// TIA Portal V19 export
VAR_GLOBAL   // PLC tag table "Default tag table"
   "HOOTER RESET" AT %Q0.0 : Bool;
   "EMERGENCY STOP" AT %I0.0 : Bool;
   "FRL LOW" AT %I0.1 : Bool;
   HOOTER AT %I0.2 : Bool;
   "MGF FEED PUMP P-101 A MCB TRIP" AT %I0.3 : Bool;
   "MGF FEED PUMP P-101 B MCB TRIP" AT %I0.4 : Bool;
   "MGF BACK WASH  P-102 A MCB TRIP" AT %I0.5 : Bool;
   "MGF BACK WASH P-102 B MCB TRIP" AT %I0.6 : Bool;
   "UF FEED PUMP P-103 A MCB TRIP" AT %I0.7 : Bool;
   "UF FEED PUMP P-103 B MCB TRIP" AT %I1.0 : Bool;
   "UF BLOWER AB-201 A MCB TRIP" AT %I1.1 : Bool;
   "UF BLOWER AB-201 B MCB TRIP" AT %I1.2 : Bool;
   "UF BACKWASH P-201A TRIP" AT %I1.3 : Bool;
   "UF BACKWASH P-201B TRIP" AT %I1.4 : Bool;
   SPARE_2 AT %I1.5 : Bool;
   "MGF FEED PUMP P-101 A" AT %Q0.1 : Bool;
   "MGF FEED PUMP P-101 B" AT %Q0.2 : Bool;
   "MGF BACK WASH P-102 A" AT %Q0.3 : Bool;
   "MGF BACK WASH P-102 B" AT %Q0.4 : Bool;
   "UF FEED PUMP P-103 A" AT %Q0.5 : Bool;
   "UF FEED PUMP P-103 B" AT %Q0.6 : Bool;
   "UF BLOWER AB-201 A" AT %Q0.7 : Bool;
   "UF BLOWER AB 201 B" AT %Q1.0 : Bool;
   "UF BACK WASH P-201 A" AT %Q1.1 : Bool;
   "SPARE(35)" AT %I8.0 : Bool;
   "SPARE(34)" AT %I8.1 : Bool;
   "DM FEED PUMP P-502 A MPCB TRIP" AT %I8.2 : Bool;
   "DM FEED PUMP P-502 B MPCB TRIP" AT %I8.3 : Bool;
   "DM FEED PUMP P-502 C MPCB TRIP" AT %I8.4 : Bool;
   "CIP P-601" AT %I8.5 : Bool;
   "BACK WASH RECOVERY P-801 A MPCB TRIP" AT %I8.6 : Bool;
   "BACK WASH RECOVERY P-801 B MPCB TRIP" AT %I8.7 : Bool;
   "ABFV-101 FEED BACK OPEN FEED BACK" AT %I9.0 : Bool;
   "ABFV-101 FEED BACK CLOSE FEED BACK" AT %I9.1 : Bool;
   "ABFV-102 FEED BACK OPEN FEED BACK" AT %I9.2 : Bool;
   "ABFV-102 FEED BACK CLOSE FEED BACK" AT %I9.3 : Bool;
   "ABFV-103 FEED BACK OPEN FEED BACK" AT %I9.4 : Bool;
   "ABFV-103 FEED BACK CLOSE FEED BACK" AT %I9.5 : Bool;
   "ABFV-104 FEED BACK OPEN FEED BACK" AT %I9.6 : Bool;
   "ABFV-104 FEED BACK CLOSE FEED BACK" AT %I9.7 : Bool;
   "UF BACK WASH  P-201 B" AT %Q8.0 : Bool;
   "DM FEED PUMP P-502 A" AT %Q8.1 : Bool;
   "DM FEED PUMP P-502 B" AT %Q8.2 : Bool;
   "DM FEED PUMP P-502 C" AT %Q8.3 : Bool;
   "CIP PUMP P-601" AT %Q8.4 : Bool;
   "BACK WASH RECOVERY P-801 A" AT %Q8.5 : Bool;
   "BACK WASH RECOVERY P-801 B" AT %Q8.6 : Bool;
   SPARE AT %Q8.7 : Bool;
   "SPARE(1)" AT %Q9.0 : Bool;
   "SPARE(2)" AT %Q9.1 : Bool;
   "DP-701" AT %Q9.2 : Bool;
   "DP-702" AT %Q9.3 : Bool;
   "NaOCL DOSING D-706 A" AT %Q9.4 : Bool;
   "NaOCL DOSING DP-706B" AT %Q9.5 : Bool;
   "ABFV-501" AT %Q9.6 : Bool;
   "ABFV-502" AT %Q9.7 : Bool;
   "ABFV 105 FEED BACK OPEN" AT %I12.0 : Bool;
   "ABFV 105 FEED BACK CLOSE" AT %I12.1 : Bool;
   "ABV 201 FEED BACK OPEN" AT %I12.2 : Bool;
   "ABV 201 FEED BACK CLOSE" AT %I12.3 : Bool;
   "ABFV 201 FEED BACK OPEN" AT %I12.4 : Bool;
   "ABFV 201 FEED BACK CLOSE" AT %I12.5 : Bool;
   "ABFV 202 FEED BACK OPEN" AT %I12.6 : Bool;
   "ABFV 202 FEED BACK CLOSE" AT %I12.7 : Bool;
   "ABFV 203 FEED BACK OPEN" AT %I13.0 : Bool;
   "ABFV 203 FEED BACK CLOSE" AT %I13.1 : Bool;
   "ABFV 204 FEED BACK OPEN" AT %I13.2 : Bool;
   "ABFV 204 FEED BACK CLOSE" AT %I13.3 : Bool;
   "ABFV 205 FEED BACK OPEN" AT %I13.4 : Bool;
   "ABFV 205 FEED BACK CLOSE" AT %I13.5 : Bool;
   "ABFV 206 FEED BACK OPEN" AT %I13.6 : Bool;
   "ABFV 206 FEED BACK CLOSE" AT %I13.7 : Bool;
   "ABFV 101 MULTIGRADE FILTER VALVE" AT %Q12.0 : Bool;
   "ABFV 102 MULTIGRADE FILTER VALVE" AT %Q12.1 : Bool;
   "ABFV 103 MULTIGRADE FILTER VALVE" AT %Q12.2 : Bool;
   "ABFV 104 MULTIGRADE FILTER VALVE" AT %Q12.3 : Bool;
   "ABFV 105 MULTIGRADE FILTER VALVE" AT %Q12.4 : Bool;
   "ABV 201 UF VALVE" AT %Q12.5 : Bool;
   "ABFV 201 UF VALVE" AT %Q12.6 : Bool;
   "ABFV 202 UF VALVE" AT %Q12.7 : Bool;
   "ABFV 203 UF VALVE" AT %Q13.0 : Bool;
   "ABFV 204 UF VALVE" AT %Q13.1 : Bool;
   "ABFV 205 UF VALVE" AT %Q13.2 : Bool;
   "ABFV 206 UF VALVE" AT %Q13.3 : Bool;
   "ABFV 207 UF VALVE" AT %Q13.4 : Bool;
   "ABFV 208 UF VALVE" AT %Q13.5 : Bool;
   "SPARE(3)" AT %Q13.6 : Bool;
   "SPARE(4)" AT %Q13.7 : Bool;
   "P-502 C ON" AT %I16.0 : Bool;
   "P-601 ON" AT %I16.1 : Bool;
   "P-801 A BACK WASH WAST FEED BACK" AT %I16.2 : Bool;
   "P-801 B BACK WASH WAST FEED BACK" AT %I16.3 : Bool;
   "SPARE(5)" AT %I16.4 : Bool;
   "SPARE(6)" AT %I16.5 : Bool;
   "SPARE(7)" AT %I16.6 : Bool;
   "SPARE(8)" AT %I16.7 : Bool;
   "SPARE(9)" AT %I17.0 : Bool;
   "SPARE(10)" AT %I17.1 : Bool;
   "ABFV 501 OPEN FEED BACK" AT %I17.2 : Bool;
   "ABFV 501 CLOSE FEED BACK" AT %I17.3 : Bool;
   "ABFV 502 OPEN FEED BACK" AT %I17.4 : Bool;
   "ABFV 502 CLOSE FEED BACK" AT %I17.5 : Bool;
   "PS 201 UF" AT %I17.6 : Bool;
   "SPARE(12)" AT %I17.7 : Bool;
   "ABFV-207 FEED BACK OPEN" AT %I18.0 : Bool;
   "ABFV-207 FEED BACK CLOSE" AT %I18.1 : Bool;
   "ABFV-208 FEED BACK OPEN" AT %I18.2 : Bool;
   "ABFV-208 FEED BACK CLOSE" AT %I18.3 : Bool;
   "P-101 A MGF FEED PUMP" AT %I18.4 : Bool;
   "P-101 B MGF FEED PUMP" AT %I18.5 : Bool;
   "P-102 A MGF BACK WASH" AT %I18.6 : Bool;
   "P-102 B MGF BACK WASH" AT %I18.7 : Bool;
   "P-103 A UF FEED PUMP" AT %I19.0 : Bool;
   "P-103 B UF FEED PUMP" AT %I19.1 : Bool;
   "AB-201 A UF BLOWER" AT %I19.2 : Bool;
   "AB-201 B UF BLOWER" AT %I19.3 : Bool;
   "P-201 A UF BACK WASH" AT %I19.4 : Bool;
   "P-201 B UF BACK WASH" AT %I19.5 : Bool;
   "P-502 A DM FEED PUMP" AT %I19.6 : Bool;
   "SPARE(13)" AT %Q16.0 : Bool;
   "UV 601" AT %Q16.1 : Bool;
   "SPARE(15)" AT %Q16.2 : Bool;
   "SPARE(16)" AT %Q16.3 : Bool;
   "SPARE(17)" AT %Q16.4 : Bool;
   "SPARE(18)" AT %Q16.5 : Bool;
   "SPARE(19)" AT %Q16.6 : Bool;
   "SPARE(20)" AT %Q16.7 : Bool;
   "SPARE(21)" AT %Q17.0 : Bool;
   "SPARE(22)" AT %Q17.1 : Bool;
   "SPARE(23)" AT %Q17.2 : Bool;
   "SPARE(24)" AT %Q17.3 : Bool;
   "SPARE(25)" AT %Q17.4 : Bool;
   "SPARE(26)" AT %Q17.5 : Bool;
   "SPARE(27)" AT %Q17.6 : Bool;
   "SPARE(28)" AT %Q17.7 : Bool;
   "LEVEL TRANSMITTER-101 ANALOG" AT %IW160 : Int;
   "LEVEL TRANSMITTER-102 ANALOG" AT %IW162 : Int;
   "DIFFRENTIAL PRESSURE TRANSMITTER-101 ANALOG" AT %IW164 : Int;
   "CONDUCTIVITY INDICATOR CUM TRANSMITTER-101" AT %IW166 : Int;
   "DIFFRENTIAL PRESSURE TRANSMITTER-201" AT %IW168 : Int;
   "FLOW INDICATIOR TOTALISER-201" AT %IW170 : Int;
   "LEVEL TRANSMITTER-201" AT %IW172 : Int;
   "LEVEL TRANSMITTER-801" AT %IW174 : Int;
   "RESISTIVITY CUM TRANSMITTER 601" AT %IW176 : Int;
   "PRESSURE TRANSMITTER 601" AT %IW178 : Int;
   "FLOW INDICATIOR TOTALISER 601" AT %IW180 : Int;
   "PH INDICATOR CUM TRANSMITTER 601" AT %IW182 : Int;
   "UV-601 SENSOR" AT %IW184 : Int;
   "SPARE(30)" AT %IW186 : Int;
   "SPARE(31)" AT %IW188 : Int;
   "SPARE(32)" AT %IW190 : Int;
   Tag_1 AT %I1.6 : Bool;
   Tag_2 AT %I10.0 : Bool;
   Tag_3 AT %I14.0 : Bool;
   "P-502 B DM FEED PUMP" AT %I19.7 : Bool;
   Tag_4 AT %Q1.2 : Bool;
   System_Byte AT %MB1 : Byte;
   FirstScan AT %M1.0 : Bool;
   DiagStatusUpdate AT %M1.1 : Bool;
   AlwaysTRUE AT %M1.2 : Bool;
   AlwaysFALSE AT %M1.3 : Bool;
   Clock_Byte AT %MB0 : Byte;
   Clock_10Hz AT %M0.0 : Bool;
   Clock_5Hz AT %M0.1 : Bool;
   "Clock_2.5Hz" AT %M0.2 : Bool;
   Clock_2Hz AT %M0.3 : Bool;
   "Clock_1.25Hz" AT %M0.4 : Bool;
   Clock_1Hz AT %M0.5 : Bool;
   "Clock_0.625Hz" AT %M0.6 : Bool;
   "Clock_0.5Hz" AT %M0.7 : Bool;
   BIT AT %M5.0 : Bool;
   UF_BIT AT %M2.0 : Bool;
   HJCHJC AT %M2.1 : Bool;
   WEWT AT %M2.2 : Bool;
   START AT %M2.3 : Bool;
   TESTING AT %M2.4 : Bool;
   "PT-601 PID NORX" AT %M6.0 : LReal;
   "PT-601 PID NOR PID" AT %M14.0 : LReal;
   "PT-601 PID NORX BAR" AT %M22.0 : LReal;
   "HMI HOOTER RESET" AT %M2.5 : Bool;
   TT AT %M2.6 : Bool;
   "HOOTER RESET HMI" AT %M2.7 : Bool;
   Tag_5 AT %IW60 : Int;
   JJJ AT %M3.0 : Bool;
   "VFD P-501A MANUAL VFD" AT %MW30 : Int;
   "VFD P-501B MANUAL VFD" AT %MW32 : Int;
   "VFD P-501C MANUAL VFD" AT %MW34 : Int;
   P_502A_PV AT %MW36 : Int;
   "ONLY_UF BACKWASH LT201 LL" AT %MW38 : Int;
END_VAR
